// SIMATIC S7-200 project (STEP 7-Micro/WIN), CPU 221 REL 01.10

ORGANIZATION_BLOCK 主程序:OB1
TITLE=程序注释
BEGIN
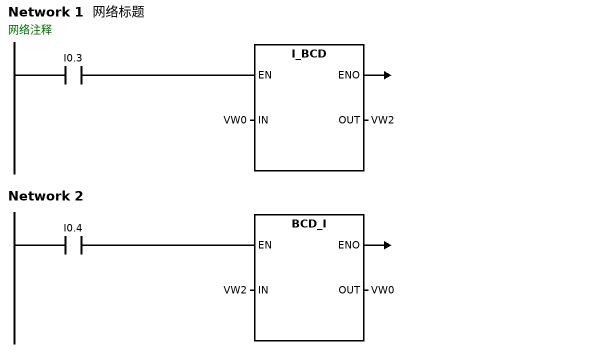
Network 1 // 网络标题
// 网络注释
LD     I0.3
MOVW   VW0, VW2
IBCD   VW2
Network 2
LD     I0.4
MOVW   VW2, VW0
BCDI   VW0
END_ORGANIZATION_BLOCK
